// Mitsubishi GX Works2 project: Project_PLC 33_Final_Version   PLC: FX3G
// project 2

// global labels: Global1
VAR_GLOBAL
  dfgdfg AT X006 : BOOL;
  awtsffg AT Y006 : BOOL;
  Start AT X007 : BOOL;
  Cream AT D1100 : REAL;
  Biscu AT D1110 : REAL;
  Choco AT D1120 : REAL;
END_VAR
VAR_GLOBAL CONSTANT
  C_lim : REAL := 300;
  B_lim : REAL := 6;
  Coco_lim : REAL := 240;
END_VAR
VAR_GLOBAL
  limitCheck AT CC1 : BOOL;
END_VAR
VAR_GLOBAL CONSTANT
  yes : INT := 1;
END_VAR
VAR_GLOBAL
  lamp_switch AT M0 : BOOL;
  Ongoing AT Y007 : BOOL;
  Yes_lim AT M0 : BOOL;
  Start_Zilof AT X010 : BOOL;
  Stop_Zilof AT X005 : BOOL;
  Zilof_On AT M4 : BOOL;
  Sen_30 AT X003 : BOOL;
  Sen_15 AT X004 : BOOL;
  Zilof_lamp AT Y004 : BOOL;
  M_Cream AT X011 : BOOL;
  Mech_Zilof AT D1102 : REAL;
END_VAR
VAR_GLOBAL CONSTANT
  Const300 : REAL := 300;
  Con0 : REAL;
END_VAR
VAR_GLOBAL
  Zilof_Finished AT M1 : BOOL;
  Zilof_Ongoing AT M4 : BOOL;
END_VAR
VAR_GLOBAL CONSTANT
  Const6 : REAL := 6;
END_VAR
VAR_GLOBAL
  TC1 AT TC1 : BOOL;
  TCS1 AT TC1 : BOOL;
END_VAR
VAR_GLOBAL CONSTANT
  W4 : INT := 4;
END_VAR
VAR_GLOBAL
  TSC1 AT TS1 : BOOL;
  Tranport1 AT Y000 : BOOL;
  TCS2 AT TC2 : BOOL;
  TSC2 AT TS2 : BOOL;
  Tranport2 AT Y001 : BOOL;
  Stop_trans AT TS7 : BOOL;
  TCC7 AT TC7 : BOOL;
END_VAR
VAR_GLOBAL CONSTANT
  W400 : INT := 400;
END_VAR
VAR_GLOBAL
  WW4 AT K30 : INT;
  Timer_tran AT M7 : BOOL;
  TCS7 AT TC7 : BOOL;
  TSC7 AT TS7 : BOOL;
  StartChoco AT X006 : BOOL;
  Type_frost AT D8280 : INT;
  frosting AT D1105 : REAL;
  less_5 AT M0 : BOOL;
END_VAR
VAR_GLOBAL CONSTANT
  K_20 : REAL := 20;
END_VAR
VAR_GLOBAL
  frost_amount AT D1130 : REAL;
END_VAR
VAR_GLOBAL CONSTANT
  K_5 : REAL := 5;
  K_40 : REAL := 40;
  K_120 : REAL := 120;
  K_240 : REAL := 240;
END_VAR
VAR_GLOBAL
  Choco_In_Process AT Y003 : BOOL;
  W5 AT K50 : INT;
  TCS8 AT TC8 : BOOL;
  Mech_Choco AT D1140 : REAL;
END_VAR
VAR_GLOBAL CONSTANT
  K_4 : REAL := 395;
END_VAR
VAR_GLOBAL
  Frost_On AT M8 : BOOL;
  TSC8 AT TS8 : BOOL;
  M_66 AT M6 : BOOL;
  M_6 AT M6 : BOOL;
  WWW4 AT K40 : INT;
  Sen_Krembo_Arrive AT X002 : BOOL;
  Sen_Camara AT X001 : BOOL;
  WW5 AT K50 : INT;
  WWWW4 AT K40 : INT;
  Singel_Pack AT X000 : BOOL;
  Counter1 AT CC1 : BOOL;
  Units AT K5 : INT;
  Almost_Finish_Pack AT Y002 : BOOL;
  OutC AT CS1 : BOOL;
  Counter2 AT CC2 : BOOL;
  Units_finish AT K6 : INT;
  Finished_Batch AT CS2 : BOOL;
  finished_Products AT D1180 : REAL;
END_VAR
VAR_GLOBAL CONSTANT
  K_1 : REAL := 1;
END_VAR
VAR_GLOBAL
  M_9 : BOOL;
  TSC9 AT TS9 : BOOL;
  WW3 AT K30 : INT;
  TCS3 AT TC3 : BOOL;
  TCS4 AT TC4 : BOOL;
  TSC3 AT TS3 : BOOL;
  TSC4 AT TS4 : BOOL;
  M_10 AT M10 : BOOL;
  OutOfResource AT M11 : BOOL;
  TCS9 AT TC9 : BOOL;
END_VAR
VAR_GLOBAL CONSTANT
  Reset : REAL;
  Dive_Const : REAL := 40;
END_VAR
VAR_GLOBAL
  Start_cool AT X001 : BOOL;
  Cool_On AT M10 : BOOL;
  Analog_Output AT D8282 : INT;
END_VAR
VAR_GLOBAL CONSTANT
  Mul_Const : REAL := 40;
END_VAR
VAR_GLOBAL
  TCS11 AT TC11 : BOOL;
  TSC11 AT TS11 : BOOL;
  WW1 AT K10 : INT;
  TCS6 AT TC6 : BOOL;
  TSC6 AT TS6 : BOOL;
  Finish_Help AT M12 : BOOL;
  WW0 AT K0 : INT;
  TCS12 AT TC12 : BOOL;
  TSC12 AT TS12 : BOOL;
  M_20 AT M20 : BOOL;
  WW6 AT K60 : INT;
  WWW6 AT K60 : INT;
  WWW_6 AT K60 : INT;
  FinsihWait AT K40 : INT;
  Finsih_Wait AT K40 : INT;
  TCS10 AT TC10 : BOOL;
  TSC10 AT TS10 : BOOL;
  WAIT AT K40 : INT;
END_VAR

// task Task_01 (event TRUE, interval 0, priority 31): POU_01

PROGRAM POU_01
(* structured ladder/FBD written out as ST: instructions are called as NAME(EN, inputs, outputs); _pN, _eN, _tN stand for wires *)
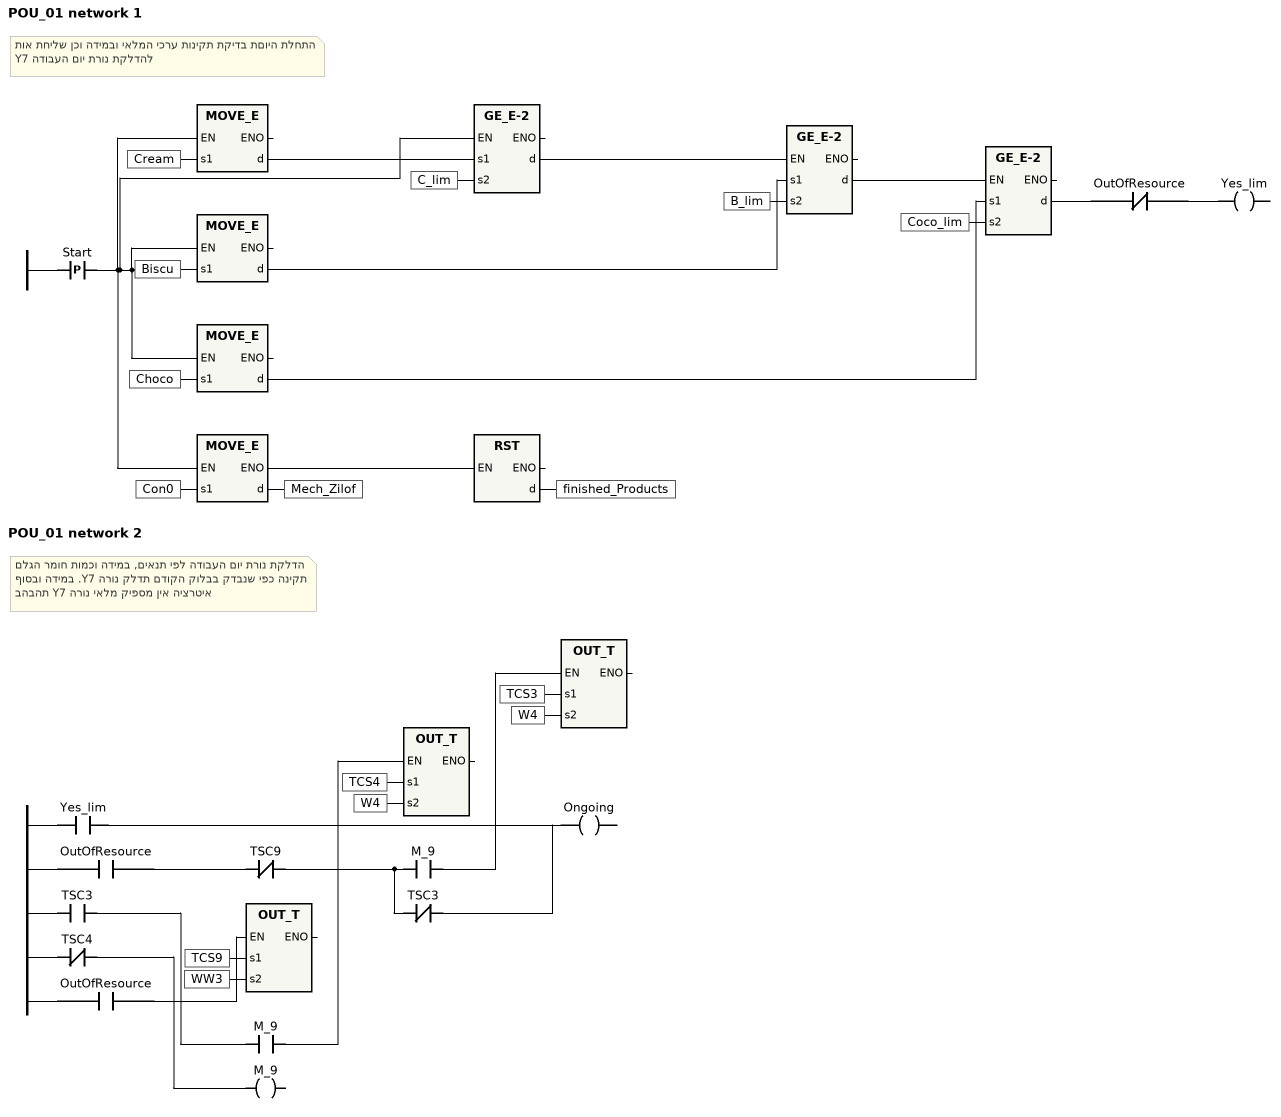
(* network 1 *)
(* התחלת היוםת בדיקת תקינות ערכי המלאי ובמידה וכן שליחת אות להדלקת נורת יום העבודה Y7 *)
_p1 := LDP(TRUE, Start);
_e2 := MOVE_E(_p1, Con0, Mech_Zilof);
RST(_e2, finished_Products);
MOVE_E(_p1, Cream, _t3);
GE_E(_p1, _t3, C_lim, _t4);
MOVE_E(_p1, Biscu, _t5);
GE_E(_t4, _t5, B_lim, _t6);
MOVE_E(_p1, Choco, _t7);
GE_E(_t6, _t7, Coco_lim, _t8);
Yes_lim := _t8 AND NOT OutOfResource;
(* network 2 *)
(* הדלקת נורת יום העבודה לפי תנאים, במידה וכמות חומר הגלם תקינה כפי שנבדק בבלוק הקודם תדלק נורה Y7. במידה ובסוף איטרציה אין מספיק מלאי נורה Y7 תהבהב *)
_p1 := OutOfResource AND NOT TSC9;
OUT_T(_p1 AND M_9, TCS3, W4);
Ongoing := Yes_lim OR (_p1 AND NOT TSC3);
OUT_T(TSC3 AND M_9, TCS4, W4);
M_9 := NOT TSC4;
OUT_T(OutOfResource, TCS9, WW3);
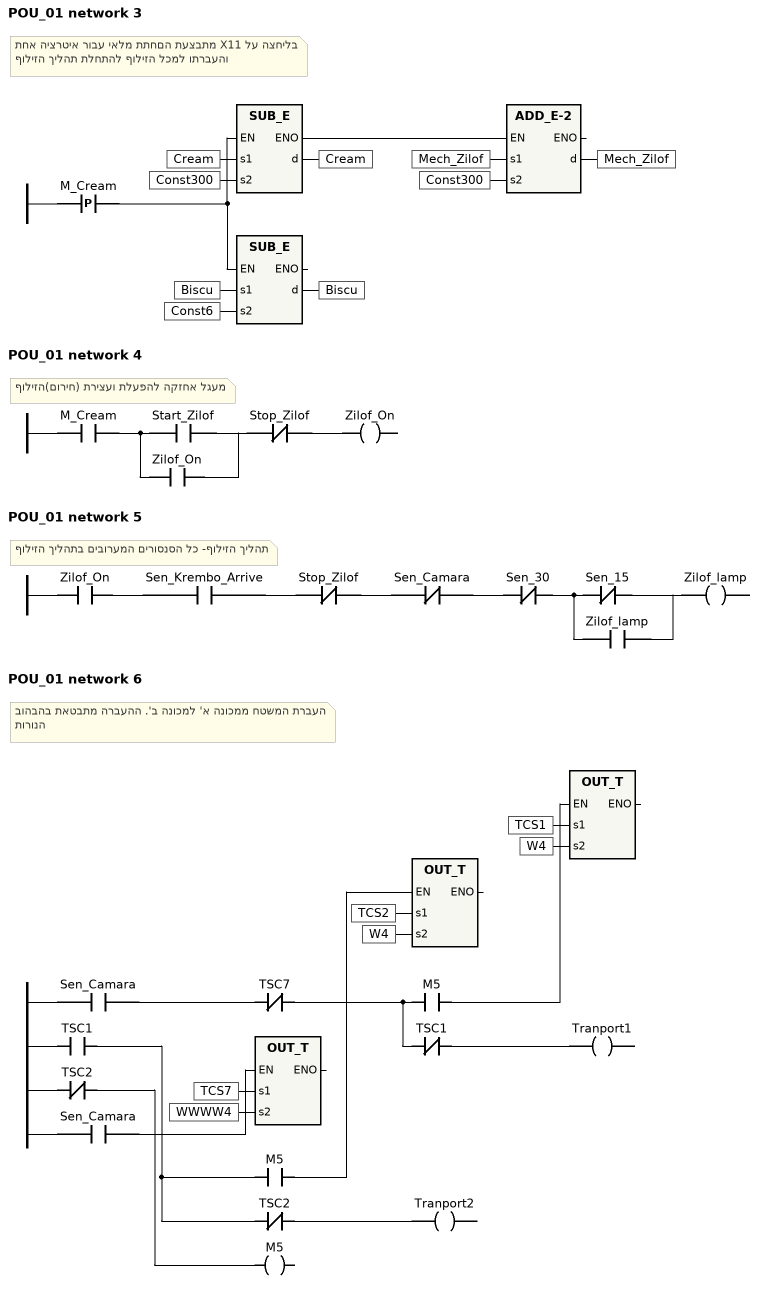
(* network 3 *)
(* בליחצה על X11 מתבצעת הםחתת מלאי עבור איטרציה אחת והעברתו למכל הזילוף להתחלת תהליך הזילוף *)
_p1 := LDP(TRUE, M_Cream);
_e2 := SUB_E(_p1, Cream, Const300, Cream);
ADD_E(_e2, Mech_Zilof, Const300, Mech_Zilof);
SUB_E(_p1, Biscu, Const6, Biscu);
(* network 4 *)
(* מעגל אחזקה להפעלת ועצירת (חירום)הזילוף *)
Zilof_On := ((M_Cream AND Start_Zilof) OR (M_Cream AND Zilof_On)) AND NOT Stop_Zilof;
(* network 5 *)
(* תהליך הזילוף- כל הסנסורים המערובים בתהליך הזילוף *)
_p1 := Zilof_On AND Sen_Krembo_Arrive AND NOT Stop_Zilof AND NOT Sen_Camara AND NOT Sen_30;
Zilof_lamp := (_p1 AND NOT Sen_15) OR (_p1 AND Zilof_lamp);
(* network 6 *)
(* העברת המשטח ממכונה א' למכונה ב'. ההעברה מתבטאת בהבהוב הנורות *)
_p1 := Sen_Camara AND NOT TSC7;
OUT_T(_p1 AND M5, TCS1, W4);
Tranport1 := _p1 AND NOT TSC1;
OUT_T(TSC1 AND M5, TCS2, W4);
Tranport2 := TSC1 AND NOT TSC2;
M5 := NOT TSC2;
OUT_T(Sen_Camara, TCS7, WWWW4);
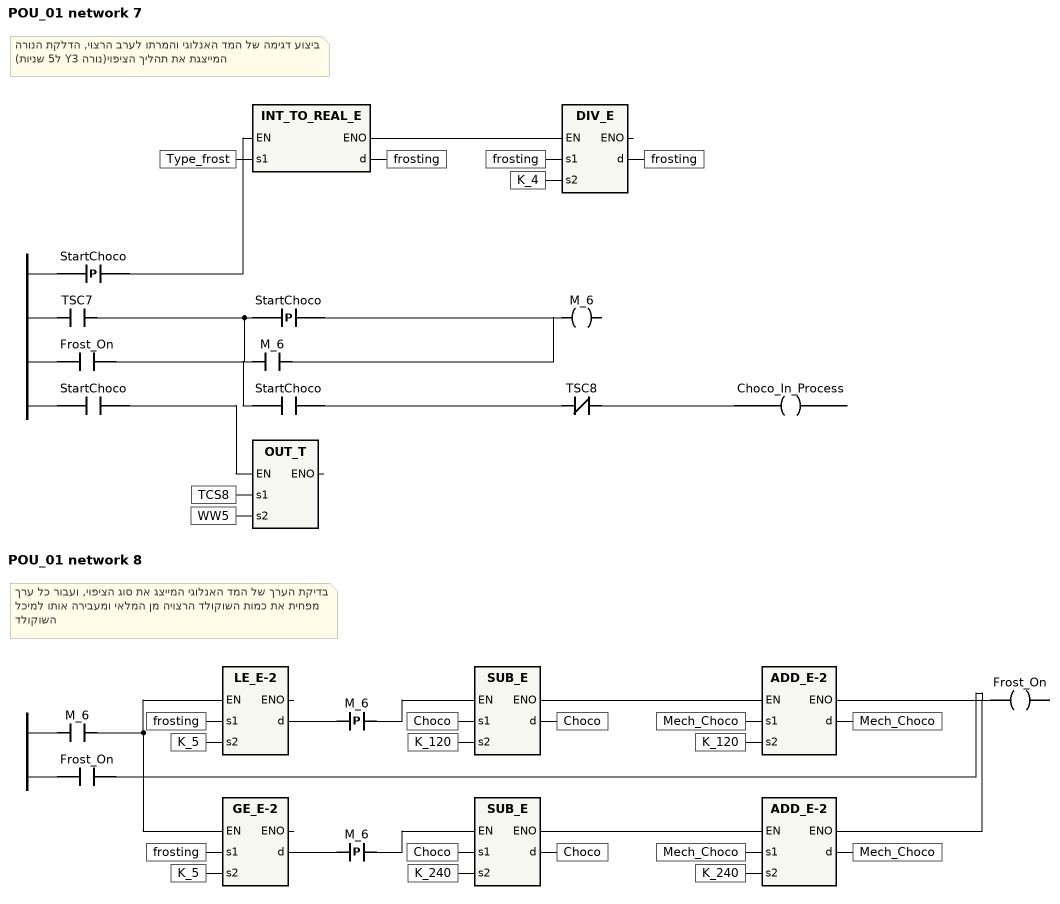
(* network 7 *)
(* ביצוע דגימה של המד האנלוגי והמרתו לערב הרצוי, הדלקת הנורה המייצגת את תהליך הציפוי(נורה Y3 ל5 שניות) *)
_e1 := INT_TO_REAL_E(LDP(TRUE, StartChoco), Type_frost, frosting);
DIV_E(_e1, frosting, K_4, frosting);
M_6 := (TSC7 AND LDP(TRUE, StartChoco)) OR (TSC7 AND M_6);
Choco_In_Process := Frost_On AND StartChoco AND NOT TSC8;
OUT_T(StartChoco, TCS8, WW5);
(* network 8 *)
(* בדיקת הערך של המד האנלוגי המייצג את סוג הציפוי, ועבור כל ערך מפחית את כמות השוקולד הרצויה מן המלאי ומעבירה אותו למיכל השוקולד *)
LE_E(M_6, frosting, K_5, _t1);
_e2 := SUB_E(_t1 AND LDP(TRUE, M_6), Choco, K_120, Choco);
_e3 := ADD_E(_e2, Mech_Choco, K_120, Mech_Choco);
GE_E(M_6, frosting, K_5, _t4);
_e5 := SUB_E(_t4 AND LDP(TRUE, M_6), Choco, K_240, Choco);
_e6 := ADD_E(_e5, Mech_Choco, K_240, Mech_Choco);
Frost_On := _e3 OR _e6 OR Frost_On;
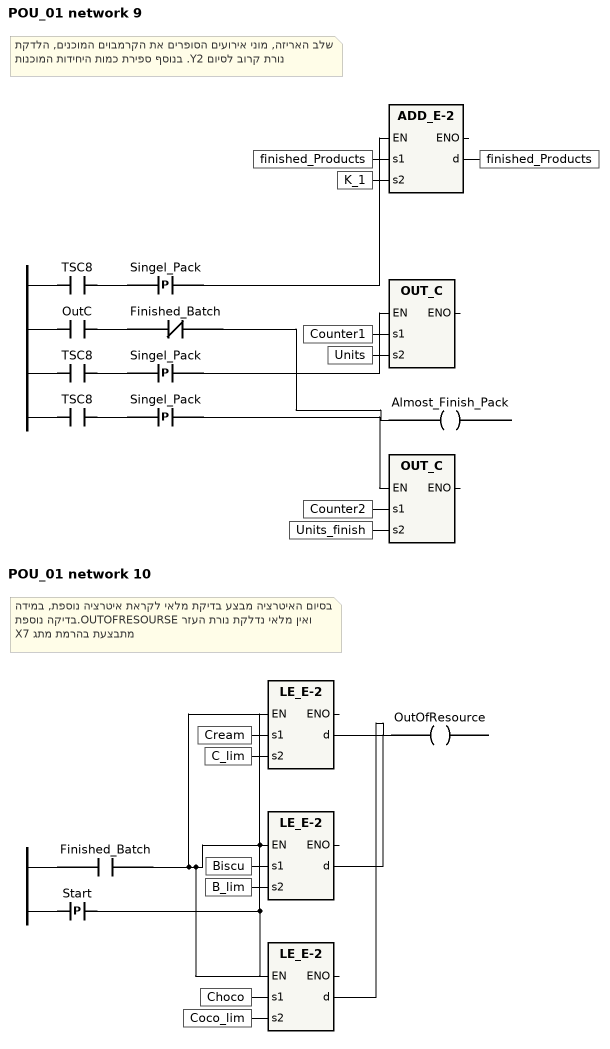
(* network 9 *)
(* שלב האריזה, מוני אירועים הסופרים את הקרמבוים המוכנים, הלדקת נורת קרוב לסיום Y2. בנוסף ספירת כמות היחידות המוכנות *)
ADD_E(TSC8 AND LDP(TRUE, Singel_Pack), finished_Products, K_1, finished_Products);
Almost_Finish_Pack := OutC AND NOT Finished_Batch;
OUT_C(TSC8 AND LDP(TRUE, Singel_Pack), Counter1, Units);
OUT_C(TSC8 AND LDP(TRUE, Singel_Pack), Counter2, Units_finish);
(* network 10 *)
(* בסיום האיטרציה מבצע בדיקת מלאי לקראת איטרציה נוספת, במידה ואין מלאי נדלקת נורת העזר OUTOFRESOURSE.בדיקה נוספת מתבצעת בהרמת מתג X7 *)
_p1 := Finished_Batch OR LDP(TRUE, Start);
LE_E(_p1, Cream, C_lim, _t2);
LE_E(_p1, Biscu, B_lim, _t3);
LE_E(_p1, Choco, Coco_lim, _t4);
OutOfResource := _t2 OR _t3 OR _t4;
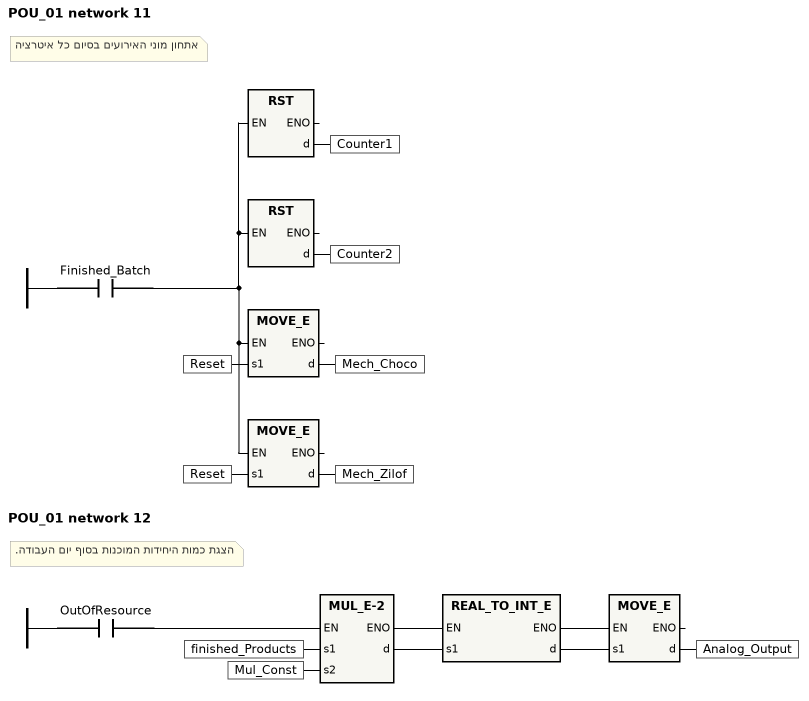
(* network 11 *)
(* אתחון מוני האירועים בסיום כל איטרציה *)
RST(Finished_Batch, Counter1);
RST(Finished_Batch, Counter2);
MOVE_E(Finished_Batch, Reset, Mech_Choco);
MOVE_E(Finished_Batch, Reset, Mech_Zilof);
(* network 12 *)
(* הצגת כמות היחידות המוכנות בסוף יום העבודה. *)
_e2 := MUL_E(OutOfResource, finished_Products, Mul_Const, _t1);
_e4 := REAL_TO_INT_E(_e2, _t1, _t3);
MOVE_E(_e4, _t3, Analog_Output);
END_PROGRAM
